INTERFACE I_Event EXTENDS __SYSTEM.IQueryInterface

END_INTERFACE

(* stored: Version 1.1.0.1, ProductVersion 3.1.4024.12
   Itf I_Event: Id {fb4af3b3-95c8-4e08-8961-bafd01f73512} *)
